FUNCTION_BLOCK FB_CRYO_PUMP_ECODRY EXTENDS FB_CRYO_PUMP_MODBUS
VAR_INPUT
END_VAR
VAR_OUTPUT
END_VAR
VAR CONSTANT
END_VAR
VAR
	{attribute 'OPC.UA.DA' := '1'}
	cfg:		T_CRYO_PUMP_MODBUS_CFG;		//  Config parameters
	{attribute 'OPC.UA.DA' := '1'}
	ctrl:		T_CRYO_PUMP_MODBUS_CTRL;	//  Control parameters
	{attribute 'OPC.UA.DA' := '1'}
	{attribute 'OPC.UA.DA.Access' := '1'}
	stat:		T_CRYO_PUMP_MODBUS_STAT;	//  Status parameters - ReadOnly


END_VAR

// Execute the base class object FB_RS_BASE
SUPER^();

METHOD M_Configure
VAR_INPUT
END_VAR
IF NOT bStarted	THEN
	//
	// START: Mandatory for ALL pumps !!!
	//
	// Set references from FB_RS_BASE
	cfgRef	REF=cfg;
	ctrlRef	REF=ctrl;
	statRef	REF=stat;

	// Set references from FB_CRYO_PUMP_BASE
	cfgBaseRef	REF=cfg;
	ctrlBaseRef	REF=ctrl;
	statBaseRef	REF=stat;

	// Set references from FB_CRYO_PUMP_MODBUS
	cfgModbusRef	REF=cfg;
	ctrlModbusRef	REF=ctrl;
	statModbusRef	REF=stat;

	// Copy input parameters to configuration
	cfg.nModel			:= in_nModel;
	cfg.bAutoMonitor	:= in_bAutoMonitor;
	cfg.tDelay_Periodic	:= DINT_TO_TIME(in_nPeriod);
	
	
	// Set pointers to arrays of commands
//	ptrInitCmds	:= ADR(cfg.cmdList_Init);(* Pointer to INIT commands *)
//	ptrReadCmds	:= ADR(cfg.cmdList_Read);(* Pointer to READ commands *)
	
	// TODO in FB that extends the functionality
	// Set pointers to comm, i.e.
	ptrCommCfg	:= ADR(comm.cfg);	(* Pointer to comm.cfg instance *)
	ptrCommCtrl	:= ADR(comm.ctrl);	(* Pointer to comm.ctrl instance *)
	ptrCommStat	:= ADR(comm.stat);	(* Pointer to comm.stat instance *)
	
	// Set comm suffixes for commands and replies
//	ptrCommCfg^.sCmdSuffix		:= '';
//	ptrCommCfg^.sReplySuffix	:= '';

	statRef.bConfigured	:= TRUE;
	bStarted			:= TRUE;
	//
	// END: Mandatory for ALL pumps !!!
	//


	// TODO USER
	// Add here real configuration
	IF in_sVersion = 'V01'	THEN
		cfg.nVersion	:= E_ECODRY_VERSION.V01;
	ELSIF in_sVersion = 'V21'  OR  in_sVersion = 'V22'	THEN
		cfg.nVersion	:= E_ECODRY_VERSION.V21_22;
	END_IF
	
	// Adjust addresses and number of words
	CASE cfg.nVersion	OF
		E_ECODRY_VERSION.V01:
			// Set register addresses
			cfg.aAddr [1]	:= 16#0040;
			cfg.aAddr [2]	:= 16#0067;
			cfg.aAddr [3]	:= 16#0667;
			cfg.aAddr [4]	:= 0;	// Unused address must be zero
			
			// Set number of words to read
			cfg.aWords [1]	:= 16;
			cfg.aWords [2]	:= 2;
			cfg.aWords [3]	:= 6;
			cfg.aWords [4]	:= 0;	// Number of words for unused address must be zero
	END_CASE
	
	cfg.nSlaveID	:= in_nSlaveID;

	
END_IF
END_METHOD

METHOD M_ExtractReadings_V01 : BOOL
VAR_INPUT
	nAddressIndex:	INT;	// Which address space to read
END_VAR
VAR
	pBuf:	POINTER TO BYTE	:= ADR(stat.nInputBuffer);
	loop:	INT;
	par:	INT;
END_VAR
// There are 3 bytes before data starts !!!
IF nAddressIndex = 1 THEN
	////////////////////////////
	// Extract Common Parameters
	////////////////////////////

	// Reference Frequency 0x40H
	// Offset 3 + 0 = 3
	stat.lrFreqRef		:= UINT_TO_LREAL(M_ByteSwapUINT(ADR(pBuf[3]))) / 100.0;
	stat.lrOutFreq		:= INT_TO_LREAL(M_ByteSwapINT(ADR(pBuf[5]))) / 100.0;
	stat.nPumpSpeed		:= LREAL_TO_DINT(stat.lrOutFreq * 60.0);	// [Hz] -> [rpm]
	stat.nMotorCurr		:= UINT_TO_DINT(M_ByteSwapUINT(ADR(pBuf[7]))) * 10;
	stat.lrOutVoltRef	:= UINT_TO_LREAL(M_ByteSwapUINT(ADR(pBuf[13]))) / 10.0;
	stat.nMotorVolt		:= UINT_TO_DINT(M_ByteSwapUINT(ADR(pBuf[15])));
	stat.lrOutPower		:= INT_TO_LREAL(M_ByteSwapINT(ADR(pBuf[17]))) / 10.0;
	
	stat.nOpTime	:= M_ByteSwapUINT(ADR(pBuf[27]));
	stat.nSwFlash	:= M_ByteSwapUINT(ADR(pBuf[29]));

	(*
	stat.lrTemperature	:= UINT_TO_LREAL(M_ByteSwapUINT(ADR(pBuf[83])));

	stat.nSwRom		:= M_ByteSwapUINT(ADR(pBuf[57]));
	stat.nNumRunCmd	:= M_ByteSwapUINT(ADR(pBuf[109]));
	stat.nFanOpTime	:= M_ByteSwapUINT(ADR(pBuf[81]));
	*)

ELSIF nAddressIndex = 2 THEN
	stat.nFanOpTime			:= M_ByteSwapUINT(ADR(pBuf[3]));
	stat.nElecTemp			:= UINT_TO_DINT(M_ByteSwapUINT(ADR(pBuf[5])));
ELSIF nAddressIndex = 3 THEN
	stat.nServiceHours		:= M_ByteSwapUINT(ADR(pBuf[3]));
	stat.nNumPumpDowns		:= M_ByteSwapUINT(ADR(pBuf[7]));
	stat.nDaysUntilService	:= M_ByteSwapUINT(ADR(pBuf[13]));
END_IF
END_METHOD

METHOD M_ExtractReadings_V21_22 : BOOL
VAR_INPUT
	nAddressIndex:	INT;	// Which address space to read
END_VAR
VAR
	pBuf:	POINTER TO BYTE	:= ADR(stat.nInputBuffer);
	loop:	INT;
	par:	INT;
END_VAR
// There are 3 bytes before data starts !!!
IF nAddressIndex = 1 THEN
	////////////////////////////
	// Extract Common Parameters
	////////////////////////////

	// Reference Frequency 0x40H
	// Offset 3 + 0 = 3
	stat.lrFreqRef		:= UINT_TO_LREAL(M_ByteSwapUINT(ADR(pBuf[3]))) / 100.0;
	stat.lrOutFreq		:= INT_TO_LREAL(M_ByteSwapINT(ADR(pBuf[5]))) / 100.0;
	stat.nMotorCurr		:= UINT_TO_DINT(M_ByteSwapUINT(ADR(pBuf[7]))) * 10;
	stat.lrOutVoltRef	:= UINT_TO_LREAL(M_ByteSwapUINT(ADR(pBuf[13]))) / 10.0;
	stat.nMotorVolt		:= UINT_TO_DINT(M_ByteSwapUINT(ADR(pBuf[15])));
	stat.lrOutPower		:= INT_TO_LREAL(M_ByteSwapINT(ADR(pBuf[17]))) / 10.0;
	
	stat.nOpTime	:= M_ByteSwapUINT(ADR(pBuf[27]));
	stat.nSwFlash	:= M_ByteSwapUINT(ADR(pBuf[29]));

	(*
	stat.lrTemperature	:= UINT_TO_LREAL(M_ByteSwapUINT(ADR(pBuf[83])));

	stat.nSwRom		:= M_ByteSwapUINT(ADR(pBuf[57]));
	stat.nNumRunCmd	:= M_ByteSwapUINT(ADR(pBuf[109]));
	stat.nFanOpTime	:= M_ByteSwapUINT(ADR(pBuf[81]));
	*)

ELSIF nAddressIndex = 2 THEN
	stat.nFanOpTime			:= M_ByteSwapUINT(ADR(pBuf[3]));
	stat.nElecTemp			:= UINT_TO_DINT(M_ByteSwapUINT(ADR(pBuf[5])));
ELSIF nAddressIndex = 3 THEN
	stat.nServiceHours		:= M_ByteSwapUINT(ADR(pBuf[3]));
	stat.nNumPumpDowns		:= M_ByteSwapUINT(ADR(pBuf[7]));
	stat.nDaysUntilService	:= M_ByteSwapUINT(ADR(pBuf[13]));
END_IF
END_METHOD

METHOD M_IsReady : BOOL
VAR_INPUT
END_VAR
//	M_UpdateStatus() sets the stat.bReady flag.
M_IsReady	:= stat.bReady;
END_METHOD

METHOD M_IsRunning : BOOL
VAR_INPUT
END_VAR
M_IsRunning	:= stat.bReady OR stat.nPumpSpeed > 0;
END_METHOD

METHOD M_ReadFromReply : BOOL
VAR_INPUT
	nAddressIndex:	INT;	// Which address space to read
END_VAR
IF cfg.nVersion	= E_ECODRY_VERSION.V01	THEN
	M_ExtractReadings_V01    (nAddressIndex);
ELSIF cfg.nVersion	= E_ECODRY_VERSION.V21_22	THEN
	M_ExtractReadings_V21_22 (nAddressIndex);
END_IF
END_METHOD

METHOD M_UpdateStatus
VAR_INPUT
END_VAR
// Update inputs
stat.bReady		:= NOT i_bRunning;	// Active low
END_METHOD

END_FUNCTION_BLOCK

(* stored: Version 1.1.0.1, ProductVersion 3.1.4024.9
   POU FB_CRYO_PUMP_ECODRY: Id {0115e2c0-2da7-4d81-bba2-c6a70950e014}, SpecialFunc None
   Method M_Configure: Id {aeab42c9-8673-4da4-8a3b-fdf4891d7fa2}
   Method M_ExtractReadings_V01: Id {14c1bce2-4514-4c1a-a2a4-833eb240c3e6}
   Method M_ExtractReadings_V21_22: Id {99aa640b-54f6-46bd-9e02-e1effac7e819}
   Method M_IsReady: Id {aead2163-e248-4f3b-9315-0c19fbfe9472}
   Method M_IsRunning: Id {99c68669-3350-41f5-b144-f23d9427a726}
   Method M_ReadFromReply: Id {59e10e37-e8b9-4a09-a551-61c44a22669b}
   Method M_UpdateStatus: Id {f3eb830f-441a-438b-a7e8-95d982d38eba} *)
